// TIA Portal project "lab10" (V15)

(* hardware
DEVICE "HMI_1"  KTP900 Basic PN
   slot 0: "HMI_1"  KTP900 Basic PN  6AV2 123-2JB03-0AX0  15.0.0.0
   slot 1: "HMI_RT_1"  KTP900 Basic PN  6AV2 123-2JB03-0AX0  15.0.0.0
   slot 5: "HMI_1.IE_CP_1"  PROFINET Interface  15.0.0.0
      slot 1: "PROFINET Interface_1"  PROFINET Interface
         slot 1: "Port_1"  Port
DEVICE "S7-1200 station_1"  S7-1200 Station
   slot 0: "Rack_0"  S7-1200 Rack  Rack  V1.0
   slot 1: "PLC_1"  CPU 1214C DC/DC/DC  6ES7 214-1AG40-0XB0  V4.2
      slot 3: "AQ 1x12BIT_1"  AQ1 signal board  6ES7 232-4HA30-0XB0  V1.0
   slot 101: "CM 1243-5"  CM 1243-5  6GK7 243-5DX30-0XE0  V1.3
   slot 102: "CM 1241 (RS485)_1"  CM 1241 (RS485)  6ES7 241-1CH30-0XB0  V1.0
*)

// ===== PLC "PLC_1"  CPU 1214C DC/DC/DC =====

VAR_GLOBAL   // PLC tag table "Default tag table"
   "START" AT %I0.0 : Bool;
   "STOP" AT %I0.1 : Bool;
   "PRACA" AT %Q0.0 : Bool;
   "AWARIA" AT %I0.7 : Bool;
   "Tag_1" AT %Q0.7 : Bool;
   "SPRZEZ" AT %M0.0 : Bool;
   "WYJSCIE_GEN" AT %Q0.3 : Bool;
   "SYG_PRACY" AT %Q0.2 : Bool;
END_VAR

DATA_BLOCK "HMI_ZMIENNE"   // DB1
{ S7_Optimized_Access := 'TRUE' }
VERSION : 0.1
   VAR
      START_HMI : Bool;
      STOP_HMI : Bool;
      TRYB_PRACY : Bool;
      ZDALNE_LOKAL : Bool;
      CZAS : Time := T#1s;
      ZWIEKSZ : Bool;
      ZMNIEJSZ : Bool;
      CZAS2 : Time := T#500ms;
   END_VAR
BEGIN
END_DATA_BLOCK

// folder: System blocks/Program resources

DATA_BLOCK "T1"   // DB2
{ S7_Optimized_Access := 'TRUE' }
AUTHOR : Simatic
FAMILY : IEC
NAME : IEC_TMR
VERSION : 1.0
// stored: InstanceOfName IEC_TIMER
"IEC_TIMER"
BEGIN
END_DATA_BLOCK

DATA_BLOCK "T2"   // DB3
{ S7_Optimized_Access := 'TRUE' }
AUTHOR : Simatic
FAMILY : IEC
NAME : IEC_TMR
VERSION : 1.0
// stored: InstanceOfName IEC_TIMER
"IEC_TIMER"
BEGIN
END_DATA_BLOCK

// folder: (top level)

ORGANIZATION_BLOCK "Main"   // OB1, LAD, ProgramCycle
TITLE = "Main Program Sweep (Cycle)"
{ S7_Optimized_Access := 'TRUE' }
VERSION : 0.1
   VAR_INPUT
      Initial_Call : Bool;   // Initial call of this OB
      Remanence : Bool;   // =True, if remanent data are available
   END_VAR
BEGIN

REGION Network 1: ZALACZANIE STEROWNIKA
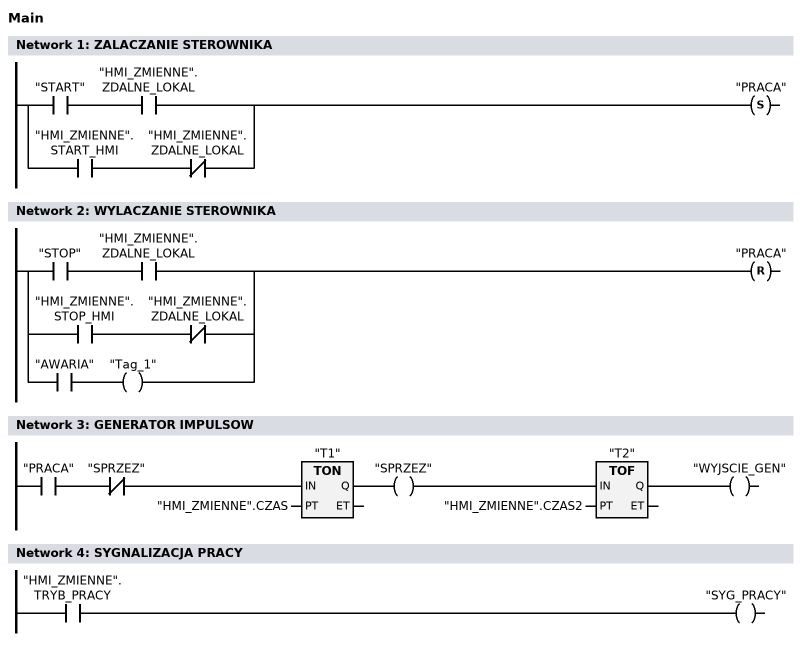
   RUNG wire#powerrail
      Contact( "START" )
      Contact( "HMI_ZMIENNE".ZDALNE_LOKAL )
      wire#w1
      S_Coil( "PRACA" )
   END_RUNG
   RUNG wire#powerrail
      Contact( "HMI_ZMIENNE".START_HMI )
      I_Contact( "HMI_ZMIENNE".ZDALNE_LOKAL )
   END_RUNG wire#w1
   // the same network as SCL:
   IF ("START" AND "HMI_ZMIENNE".ZDALNE_LOKAL) OR ("HMI_ZMIENNE".START_HMI AND NOT "HMI_ZMIENNE".ZDALNE_LOKAL) THEN
       "PRACA" := TRUE;
   END_IF;
END_REGION

REGION Network 2: WYLACZANIE STEROWNIKA
   RUNG wire#powerrail
      Contact( "STOP" )
      Contact( "HMI_ZMIENNE".ZDALNE_LOKAL )
      wire#w1
      R_Coil( "PRACA" )
   END_RUNG
   RUNG wire#powerrail
      Contact( "HMI_ZMIENNE".STOP_HMI )
      I_Contact( "HMI_ZMIENNE".ZDALNE_LOKAL )
   END_RUNG wire#w1
   RUNG wire#powerrail
      Contact( "AWARIA" )
      Coil( "Tag_1" )
   END_RUNG wire#w1
   // the same network as SCL:
   "Tag_1" := "AWARIA";
   IF ("STOP" AND "HMI_ZMIENNE".ZDALNE_LOKAL) OR ("HMI_ZMIENNE".STOP_HMI AND NOT "HMI_ZMIENNE".ZDALNE_LOKAL) OR "AWARIA" THEN
       "PRACA" := FALSE;
   END_IF;
END_REGION

REGION Network 3: GENERATOR IMPULSOW
   "T1".TON(IN := "PRACA" AND NOT "SPRZEZ", PT := "HMI_ZMIENNE".CZAS);
   "SPRZEZ" := "T1".Q;
   "T2".TOF(IN := "T1".Q, PT := "HMI_ZMIENNE".CZAS2);
   "WYJSCIE_GEN" := "T2".Q;
END_REGION

REGION Network 4: SYGNALIZACJA PRACY
   RUNG wire#powerrail
      Contact( "HMI_ZMIENNE".TRYB_PRACY )
      Coil( "SYG_PRACY" )
   END_RUNG
   // the same network as SCL:
   "SYG_PRACY" := "HMI_ZMIENNE".TRYB_PRACY;
END_REGION
END_ORGANIZATION_BLOCK

(* ===== HMI "HMI_RT_1" =====
system functions are stored by id; their names below are inferred from use
connection "HMI_Connection_1": ETHERNET, SMART_S7_1200_OMS

HMI tags "Default tag table"
   "HMI_ZMIENNE_START_HMI" : Bool = PLC HMI_ZMIENNE.START_HMI, 1 s
   "HMI_ZMIENNE_STOP_HMI" : Bool = PLC HMI_ZMIENNE.STOP_HMI, 1 s
   "HMI_ZMIENNE_TRYB_PRACY" : Bool = PLC HMI_ZMIENNE.TRYB_PRACY, 1 s
   "HMI_ZMIENNE_ZDALNE_LOKAL" : Bool = PLC HMI_ZMIENNE.ZDALNE_LOKAL, 1 s
   "PRACA" : Bool = PLC PRACA AT %Q0.0, 1 s
   "AWARIA" : Bool = PLC AWARIA AT %I0.7, 1 s
   "HMI_ZMIENNE_CZAS" : Time = PLC HMI_ZMIENNE.CZAS, 1 s
   "HMI_ZMIENNE_CZAS2" : Time = PLC HMI_ZMIENNE.CZAS2, 1 s

screen "sterowanie" 800x480
   Circle "Circle_4" at 100,135 size 53x53
      Appearance <- "PRACA"
   TextField "Text field_1" at 84,96 size 101x20; Text 'SYGNALIZACJA'
   TextField "Text field_2" at 181,152 size 50x20; Text 'PRACA'
   TextField "Text field_3" at 184,232 size 52x20; Text 'POSTÓJ'
   TextField "Text field_4" at 184,315 size 62x20; Text 'AWARIA'
   TextField "Text field_5" at 621,95 size 88x20; Text 'STEROWANIE'
   Button "Button_1" at 622,147 size 96x32; TextOff 'START'
      on Press: function_b14e0dd5("HMI_ZMIENNE_START_HMI", 0)
   Button "Button_2" at 620,201 size 96x32; TextOff 'STOP'
      on Press: function_b14e0dd5("HMI_ZMIENNE_STOP_HMI", 0)
   Switch "Switch_1" at 619,321 size 97x32; CaptionText 'Switch'; TextOff 'OFF'; TextOn 'ON'
      ProcessValue <- "HMI_ZMIENNE_ZDALNE_LOKAL"
   TextField "Text field_6" at 61,33 size 90x20; Text 'STANOWISKO'
   Circle "Circle_1" at 100,219 size 53x53
      Appearance <- "PRACA"
   Circle "Circle_2" at 99,300 size 53x53
      Appearance <- "AWARIA"
   Button "Button_3" at 620,272 size 96x32; TextOff 'TRYB'
      on Press: InvertBit("HMI_ZMIENNE_TRYB_PRACY")
   Button "Button_4" at 613,419 size 96x32; TextOff '>>'
      on Change: ActivateScreen("parametryzacja", 0)

screen "parametryzacja" 800x480
   Button "Button_1" at 25,425 size 96x32; TextOff '<<'
      on Change: ActivateScreen("sterowanie", 0)
   IOField "I/O field_1" at 180,51 size 96x32; FormatPattern s9999999999
      ProcessValue <- "HMI_ZMIENNE_CZAS"
   IOField "I/O field_3" at 180,100 size 96x32; FormatPattern s9999999999
      ProcessValue <- "HMI_ZMIENNE_CZAS2"
   TextField "Text field_1" at 128,6 size 171x20; Text 'NASTAWA GENERATOROW'
   TextField "Text field_2" at 118,51 size 46x20; Text 'OKRES'
   TextField "Text field_3" at 73,100 size 89x20; Text 'WYPELNIENIE'
*)